(* PLC project AstraRegul_stand.project, Prosoft-Systems Ltd. Astra.IDE Astra.IDE V1.7.0.0 *)
(* stored: creationDateTime 2023-10-03T18:26:20.333407, modificationDateTime 2023-09-05T16:47:00.711365 *)

FUNCTION FC_StopDone : DWORD
  VAR_IN_OUT
    EventPrm : CmpApp.EVTPARAM_CmpAppStop;
  END_VAR

                    IS_ACTIVE := FALSE;
IS_CPU_A := FALSE;
IS_CPU_B := FALSE;

                  
END_FUNCTION

FUNCTION FC_Exception : DWORD
  VAR_IN_OUT
    EventPrm : CmpApp.EVTPARAM_CmpAppException;
  END_VAR

                    IS_ACTIVE := FALSE;
IS_CPU_A := FALSE;
IS_CPU_B := FALSE;

                  
END_FUNCTION

PROGRAM MAIN
  VAR
    FB_AI1 : PsTechEE.AI1;
    FB_MODEL_VLV_C2 : PsTechEE.MODEL_VLV_C2;
    FB_VLV_C2 : PsTechEE.VLV_C2;
    FB_MODEL_VLV_D : PsTechEE.MODEL_VLV_D;
    FB_VLV_D : PsTechEE.VLV_D;
  END_VAR

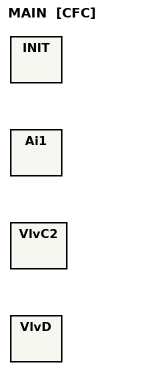
(* CFC diagram, written out as Structured Text *)
INIT();
Ai1();
VlvC2();
VlvD();

ACTION Ai1:
(* CFC diagram, written out as Structured Text *)
FB_AI1(IN := MODULE_AI_08_041.CH01.VALUE, CH_FAULT := MODULE_AI_08_041.CH01.STATUS.7, MODULFAULT := AI_08_041.HwError, SIGN_OFF := GVL.Ai1SignOff, MAN_ON := GVL.Ai1MainOn, MAN_VALUE := GVL.Ai1MainValue);
(* drawn but not wired to any output: 4, TRUE, 20, GVL.Ai1Ymin, GVL.Ai1Ymax, 3.5, 21, GVL.Ai1Tf, GVL.Ai1Ah2, GVL.Ai1Ah, GVL.Ai1Wh, GVL.Ai1Wl, GVL.Ai1Al, GVL.Ai1Al2, GVL.Ai1Hyst, GVL.Ai1SignCheck *)
END_ACTION

ACTION VlvC2:
(* CFC diagram, written out as Structured Text *)
FB_MODEL_VLV_C2(RUNTIME := GVL.VlvC2Runtime - 1, STARTTIME := 1.0, PRESSTIME := 1.0);
GVL.VlvC2Pi := FB_MODEL_VLV_C2.PI;
FB_VLV_C2(HMI_CMD := GVL.VlvC2HmiCmd, SET_MODE := GVL.VlvC2Mode, PI := GVL.VlvC2Pi);
(* drawn but not wired to any output: FALSE, GVL.VlvC2Runtime, 1.0, PsTechEE.ENUM_VALVE_FAILACTION.STP, PsTechEE.ENUM_TYPECTL.POTENT, FALSE, 2, 3.0, FALSE, 3.0, 2, 5.0, 3.0, FALSE, FALSE, FB_MODEL_VLV_C2.POWER.VALUE *)
END_ACTION

ACTION GetDefault:
                        	GetDefaultFlag	:= TRUE;

	Ai1Hyst			:= 1;
	Ai1Ymin			:= 0;
	Ai1Ymax			:= 100;
	Ai1Tf			:= 2;
	Ai1Ah			:= 90;
	Ai1Ah2			:= 95;
	Ai1Wh			:= 75;
	Ai1Wl			:= 10;
	Ai1Al			:= 5;
	Ai1Al2			:= 2;
	
	VlvC2Runtime	:= 25.0;
                      
END_ACTION

ACTION Init:
                        IF GetDefaultFlag THEN
	GetDefault();
	GetDefaultFlag := FALSE;
END_IF
                      
END_ACTION

ACTION VlvD:
(* CFC diagram, written out as Structured Text *)
FB_MODEL_VLV_D(VALVE_TYPE := 1, MOVECNT_TYPE := 0);
FB_VLV_D(HMI_CMD := Gvl.VlvDHmiCmd, SET_MODE := Gvl.VlvDMode);
(* drawn but not wired to any output: TRUE, Gvl.VlvDOpnTime, Gvl.VlvDClsTime, 2, 2, 3, FALSE, FB_MODEL_VLV_D.POWER.VALUE *)
END_ACTION
END_PROGRAM

PROGRAM DIAGN

                    REDUNDANCY();
R500_Crate();

                  

ACTION REDUNDANCY:
                        //Режим резервирования
RED_MODE := PsRedundancy_OS.GetMode();

//Активный ПЛК
IS_ACTIVE := (RED_MODE = PsRedundancy_OS.ACTIVE_STANDALONE) OR (RED_MODE = PsRedundancy_OS.ACTIVE);

//ПЛК А
IS_CPU_A := PsRedundancy_OS.IsCpuA();

//ПЛК В
IS_CPU_B := NOT IS_CPU_A;

//Синхронизация
PsRedundancy_OS.GetSyncTaskStat(SYNC_STATE);

                      
END_ACTION

ACTION R500_Crate:
                        PsDiagn.PROXY_ST_01_012(MODULE := ST_xx_x1x, DATA := MODULE_ST_xx_x1x);
PsDiagn.PROXY_PP_00_011(MODULE := PP_00_xxx, DATA := MODULE_PP_00_xxx);
PsDiagn.GET_CPU_INFO_R500(REGULBUS_HW := Regul_Bus_OS.HwError, SYNC_OK := SYNC_STATE.SyncStat.SyncOk, HW := CU_00_xxx.HwError, PF := FALSE, INFO => MODULE_CU_00_xxx);
PsDiagn.PROXY_AI_08_041(MODULE := AI_08_041, DATA := MODULE_AI_08_041);
PsDiagn.PROXY_DI_32_011(MODULE := DI_32_011, DATA := MODULE_DI_32_011);
PsDiagn.PROXY_AO_08_031(MODULE := AO_08_031, DATA := MODULE_AO_08_031);
PsDiagn.PROXY_DO_32_011(MODULE := DO_32_011, DATA := MODULE_DO_32_011);
PsDiagn.PROXY_DA_03_011_ENC(MODULE := DA_03_011, DATA := MODULE_DA_03_011);
PsDiagn.PROXY_ST_01_022(MODULE := ST_xx_x2x, DATA := MODULE_ST_xx_x2x);

                      
END_ACTION
END_PROGRAM

FUNCTION FC_PrepareShutdown : DWORD
  VAR_IN_OUT
    EventPrm : Component_Manager.EVTPARAM_CmpMgr_Shutdown;
  END_VAR

                    IS_ACTIVE := FALSE;
IS_CPU_A := FALSE;
IS_CPU_B := FALSE;

                  
END_FUNCTION

CONFIGURATION REGUL_R500_71_W
  RESOURCE Application ON PLC
    {attribute 'symbol' := 'readwrite'}
    VAR_GLOBAL  (* GVL_DIAGN *)
      IS_ACTIVE : BOOL;  (* Флаг активности ПЛК *)
      IS_CPU_A : BOOL;  (* Активность ПЛК А *)
      IS_CPU_B : BOOL;  (* Активность ПЛК Б *)
      RED_MODE : PsRedundancy_OS.RedMode;  (* Режим резервирования ПЛК *)
      SYNC_STATE : PsRedundancy_OS.TSyncTaskStat;  (* Состояние синхронизации проектов *)
      MODULE_ST_xx_x1x : PsDiagn.MODULE_ST_01_012;
      MODULE_PP_00_xxx : PsDiagn.MODULE_PP_00_011;
      MODULE_CU_00_xxx : PsDiagn.MODULE_CU_XX_XXX;
      MODULE_AI_08_041 : PsDiagn.MODULE_AI_08_041;
      MODULE_DI_32_011 : PsDiagn.MODULE_DI_32_011;
      MODULE_AO_08_031 : PsDiagn.MODULE_AO_08_031;
      MODULE_DO_32_011 : PsDiagn.MODULE_DO_32_011;
      MODULE_DA_03_011 : PsDiagn.MODULE_DA_03_011_ENC;
      MODULE_ST_xx_x2x : PsDiagn.MODULE_ST_01_022;
    END_VAR
    {attribute 'symbol' := 'readwrite'}
    VAR_GLOBAL  (* GVL - {attribute 'qualified_only'} *)
      GetDefaultFlag : BOOL;
      Ai1SignOff : BOOL;
      Ai1MainOn : BOOL;
      Ai1MainValue : REAL;
      Ai1Hyst : REAL;
      Ai1Ymin : REAL;
      Ai1Ymax : REAL;
      Ai1Tf : REAL;
      Ai1Ah : REAL;
      Ai1Ah2 : REAL;
      Ai1Wh : REAL;
      Ai1Wl : REAL;
      Ai1Al : REAL;
      Ai1Al2 : REAL;
      Ai1SignCheck : WORD;
      VlvC2Runtime : REAL;
      VlvC2Mode : PsTechEE.ENUM_MODE;
      VlvC2HmiCmd : WORD;
      VlvC2Pi : PsTechEE.AI;
      VlvDOpnTime : REAL;
      VlvDClsTime : REAL;
      VlvDHmiCmd : WORD;
      VlvDMode : PsTechEE.ENUM_MODE;
    END_VAR
    TASK MAIN_TASK(INTERVAL := T#100ms, PRIORITY := 1);
    TASK TASK_DIAGN(INTERVAL := T#1000ms, PRIORITY := 10);
    PROGRAM MAIN WITH MAIN_TASK : MAIN;
    PROGRAM DIAGN WITH TASK_DIAGN : DIAGN;
  END_RESOURCE
END_CONFIGURATION

CONFIGURATION Regul_Bus_OS
END_CONFIGURATION

CONFIGURATION R500_Crate
END_CONFIGURATION

CONFIGURATION ST_xx_x1x
END_CONFIGURATION

CONFIGURATION PP_00_xxx
END_CONFIGURATION

CONFIGURATION CU_00_xxx
END_CONFIGURATION

CONFIGURATION AI_08_041
END_CONFIGURATION

CONFIGURATION DI_32_011
END_CONFIGURATION

CONFIGURATION AO_08_031
END_CONFIGURATION

CONFIGURATION DO_32_011
END_CONFIGURATION

CONFIGURATION DA_03_011
END_CONFIGURATION

CONFIGURATION ST_xx_x2x
END_CONFIGURATION
